ABB RobotStudio station: 1660_smart_tool_trial_final_i_hope - Copy.rsstn

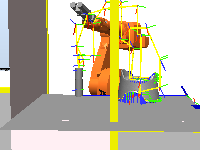
Station 1660_smart_tool_trial_final_i_hope (saved by RobotStudio format 3)
Controller 16-63074
  mechanical unit ROB_1: IRB1600_6_120__02, 6 joints, base frame (0, 0, 0) mm
Layout (positions relative to the parent item):
  - IRB1600_6_120__02 [mechanism, from Robots\IRB1600_6_120__02.rslib] at (0, 0, 0) mm; joint values [-2.0086, -0.3088, 0.1754, -0.2454, -0.2574, 6.5257] (rad or m)
  - Table [part] at (-604.56, -1688.55, 511.81) mm
  - potty-raw7 [part] at (247.23, -520.05, 664.68) mm, rotated rx 89.84 ry 0 rz 0 deg
  - holder [part, from Libraries\holder.rslib] at (-339.39, -762.82, 513.51) mm
  - Dist_to_holder [part] at (-363.16, -741.72, 512.9) mm
  - SmartComponent_1 [smart component] at (-276.35, -599.89, 1043.13) mm, rotated rx -2.86 ry 68.05 rz -114.34 deg
      signals: DI GripperClose, DI GripperOpen
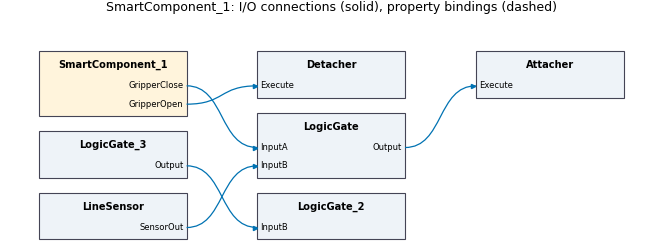
      connections:
        SmartComponent_1.GripperClose -> LogicGate.InputA
        LogicGate.Output -> Attacher.Execute
        LogicGate_3.Output -> LogicGate_2.InputB
        LineSensor.SensorOut -> LogicGate.InputB
        SmartComponent_1.GripperOpen -> Detacher.Execute
    - Kosy_Tool_No_Pen [mechanism] at (0, 0, 0) mm
        TCP Kosy_Tool_No_Pen at (121, 0, 178) mm
        links: tool-m2
    - Attacher [smart component, from Components\Attacher.rslib]
        properties: Parent=Kosy_Tool_No_Pen; Flange=0; Child=tool-m2; Mount=false; Offset=[0 0 0]; Orientation=[0 0 0]
    - Detacher [smart component, from Components\Detacher.rslib]
        properties: Child=tool-m2; KeepPosition=true
    - LogicGate [smart component, from Components\LogicGate.rslib]
        properties: Operator=AND; Delay=0
    - LogicGate_2 [smart component, from Components\LogicGate.rslib]
        properties: Operator=AND; Delay=0
    - LogicGate_3 [smart component, from Components\LogicGate.rslib]
        properties: Operator=NOT; Delay=0
    - LineSensor [smart component, from Components\LineSensor.rslib] at (-8.98, 1.66, 185.12) mm, rotated rx 90 ry 0 rz 90 deg
        properties: Start=[0 0 0]; End=[0 0 0.02]; Radius=0.004; SensedPart=(none); SensedPoint=[0 0 0]
      - _sensorPart_ [part]
  - tool-m2 [part] at (-413.78, -599.19, 679.79) mm, rotated rx -89.18 ry -2.32 rz -154.99 deg
  - Dist_to_backwall [part] at (0, -688.26, 499.44) mm
  - backwall [part] at (-1365.47, 1257.61, -1429.17) mm, rotated rx 90 ry 0 rz 0 deg
  - side wall [part] at (-604.66, -1489.36, -1403.01) mm, rotated rx 90 ry 0 rz 90 deg
  - Dist_to_sidewall2 [part] at (333.28, -1279.39, 533.83) mm
  - sidewall2 [part] at (1386.65, -1478.12, -1427.79) mm, rotated rx 0 ry -90 rz 0 deg
  - Fence_2500 [graphiccomponentgroup, from Equipment\Fence_2500.rslib] at (-617.42, -469.44, -409.13) mm, rotated rx 0 ry 0 rz 90 deg
    - Body 1 [part, from Equipment\Fence_2500.rslib]
    - Body 2 [part, from Equipment\Fence_2500.rslib]
  - bottom [part] at (306.66, -1495.49, -398.13) mm, rotated rx 0 ry -90 rz 90 deg
  - Gate [graphiccomponentgroup, from Equipment\Fence_Gate.rslib] at (-98.47, -1503.2, -434.3) mm, rotated rx 0 ry 0 rz -90 deg
    - Body 1 [part, from Equipment\Fence_Gate.rslib]
    - Body 2 [part, from Equipment\Fence_Gate.rslib]
    - Body 3 [part, from Equipment\Fence_Gate.rslib]
  - ground [part] at (-4365.19, -3484.91, 5.92) mm
Attachment: SmartComponent_1 is attached to IRB1600_6_120__02 / Link6
Collision set CollisionSet_1: SmartComponent_1, tool-m2 against Table, bottom, backwall, Fence_2500, Gate, sidewall2, side wall, near miss 0.005 m
Station logic (signal -> signal, property => property):
  16-63074.OpenGripper -> SmartComponent_1.GripperOpen
  16-63074.CloseGripper -> SmartComponent_1.GripperClose
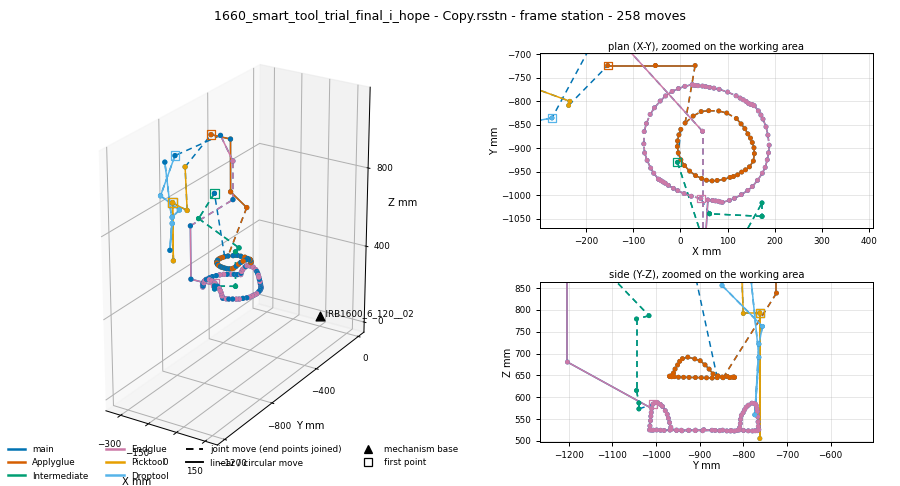
[picture p0: tool path of 1660_smart_tool_trial_final_i_hope - Copy.rsstn in frame station, 258 of 258 moves have a stored position in this frame; points joined in program order, loops and branches not executed]
Targets, tools, work objects and paths stored in the station, written as RAPID:
! task T_ROB1
MODULE MainModule
  TASK PERS tooldata tool1:=[TRUE,[[120.656,0.177793,177.769],[1,0,0,0]],[2,[0,50,88],[1,0,0,0],0,0,0]];
  PROC main()
    MoveJ Target_1290,v600,z100,Kosy_Tool\WObj:=Kosy_wobj;
    MoveJ Target_1210,v600,z100,Kosy_Tool\WObj:=Kosy_wobj;
    WaitTime 1;
    MoveJ Target_1200,v600,z100,Kosy_Tool\WObj:=Kosy_wobj;
    MoveJ Target_1190,v600,z100,Kosy_Tool\WObj:=Kosy_wobj;
    MoveJ Target_1180,v600,z100,Kosy_Tool\WObj:=Kosy_wobj;
    MoveJ Target_360,v600,z100,Kosy_Tool\WObj:=Kosy_wobj;
    MoveL Target_370,v600,z100,Kosy_Tool\WObj:=Kosy_wobj;
    MoveL Target_380,v600,z100,Kosy_Tool\WObj:=Kosy_wobj;
    MoveL Target_390,v600,z100,Kosy_Tool\WObj:=Kosy_wobj;
    MoveJ Target_10,v500,z100,Kosy_Tool\WObj:=Kosy_wobj;
    MoveJ Target_20,v500,z100,Kosy_Tool\WObj:=Kosy_wobj;
    MoveJ Target_30,v500,z100,Kosy_Tool\WObj:=Kosy_wobj;
    MoveJ Target_40,v500,z100,Kosy_Tool\WObj:=Kosy_wobj;
    MoveJ Target_50,v500,z100,Kosy_Tool\WObj:=Kosy_wobj;
    MoveJ Target_60,v500,z100,Kosy_Tool\WObj:=Kosy_wobj;
    MoveJ Target_70,v500,z100,Kosy_Tool\WObj:=Kosy_wobj;
    MoveJ Target_80,v500,z100,Kosy_Tool\WObj:=Kosy_wobj;
    MoveJ Target_90,v500,z100,Kosy_Tool\WObj:=Kosy_wobj;
    MoveJ Target_100,v500,z100,Kosy_Tool\WObj:=Kosy_wobj;
    MoveJ Target_110,v500,z100,Kosy_Tool\WObj:=Kosy_wobj;
    MoveJ Target_120,v500,z100,Kosy_Tool\WObj:=Kosy_wobj;
    MoveJ Target_130,v500,z100,Kosy_Tool\WObj:=Kosy_wobj;
    MoveJ Target_140,v500,z100,Kosy_Tool\WObj:=Kosy_wobj;
    MoveJ Target_150,v500,z100,Kosy_Tool\WObj:=Kosy_wobj;
    MoveJ Target_160,v500,z100,Kosy_Tool\WObj:=Kosy_wobj;
    MoveJ Target_170,v500,z100,Kosy_Tool\WObj:=Kosy_wobj;
    MoveJ Target_180,v500,z100,Kosy_Tool\WObj:=Kosy_wobj;
    MoveJ Target_190,v500,z100,Kosy_Tool\WObj:=Kosy_wobj;
    MoveJ Target_200,v500,z100,Kosy_Tool\WObj:=Kosy_wobj;
    MoveJ Target_210,v500,z100,Kosy_Tool\WObj:=Kosy_wobj;
    MoveJ Target_220,v500,z100,Kosy_Tool\WObj:=Kosy_wobj;
    MoveJ Target_230,v500,z100,Kosy_Tool\WObj:=Kosy_wobj;
    MoveJ Target_240,v500,z100,Kosy_Tool\WObj:=Kosy_wobj;
    MoveJ Target_250,v500,z100,Kosy_Tool\WObj:=Kosy_wobj;
    MoveJ Target_260,v500,z100,Kosy_Tool\WObj:=Kosy_wobj;
    MoveJ Target_270,v500,z100,Kosy_Tool\WObj:=Kosy_wobj;
    MoveJ Target_280,v500,z100,Kosy_Tool\WObj:=Kosy_wobj;
    MoveJ Target_290,v500,z100,Kosy_Tool\WObj:=Kosy_wobj;
    MoveJ Target_300,v500,z100,Kosy_Tool\WObj:=Kosy_wobj;
    MoveJ Target_310,v500,z100,Kosy_Tool\WObj:=Kosy_wobj;
    MoveJ Target_320,v500,z100,Kosy_Tool\WObj:=Kosy_wobj;
    MoveJ Target_330,v500,z100,Kosy_Tool\WObj:=Kosy_wobj;
    MoveJ Target_340,v500,z100,Kosy_Tool\WObj:=Kosy_wobj;
    MoveJ Target_350,v500,z100,Kosy_Tool\WObj:=Kosy_wobj;
    MoveJ Target_400,v600,z100,Kosy_Tool\WObj:=Kosy_wobj;
    MoveJ Target_410,v600,z100,Kosy_Tool\WObj:=Kosy_wobj;
    MoveJ Target_420,v600,z100,Kosy_Tool\WObj:=Kosy_wobj;
    MoveJ Target_430,v600,z100,Kosy_Tool\WObj:=Kosy_wobj;
    MoveJ Target_440,v600,z100,Kosy_Tool\WObj:=Kosy_wobj;
    MoveJ Target_450,v600,z100,Kosy_Tool\WObj:=Kosy_wobj;
    MoveJ Target_460,v600,z100,Kosy_Tool\WObj:=Kosy_wobj;
    MoveJ Target_470,v500,z100,Kosy_Tool\WObj:=Kosy_wobj;
    MoveJ Target_480,v500,z100,Kosy_Tool\WObj:=Kosy_wobj;
    MoveJ Target_490,v500,z100,Kosy_Tool\WObj:=Kosy_wobj;
    MoveJ Target_500,v500,z100,Kosy_Tool\WObj:=Kosy_wobj;
    MoveJ Target_510,v500,z100,Kosy_Tool\WObj:=Kosy_wobj;
    MoveJ Target_520,v500,z100,Kosy_Tool\WObj:=Kosy_wobj;
    MoveJ Target_530,v500,z100,Kosy_Tool\WObj:=Kosy_wobj;
    MoveJ Target_540,v500,z100,Kosy_Tool\WObj:=Kosy_wobj;
    MoveJ Target_550,v500,z100,Kosy_Tool\WObj:=Kosy_wobj;
    MoveJ Target_560,v500,z100,Kosy_Tool\WObj:=Kosy_wobj;
    MoveJ Target_570,v500,z100,Kosy_Tool\WObj:=Kosy_wobj;
    MoveJ Target_580,v500,z100,Kosy_Tool\WObj:=Kosy_wobj;
    MoveJ Target_590,v500,z100,Kosy_Tool\WObj:=Kosy_wobj;
    MoveJ Target_600,v500,z100,Kosy_Tool\WObj:=Kosy_wobj;
    MoveJ Target_610,v500,z100,Kosy_Tool\WObj:=Kosy_wobj;
    MoveJ Target_620,v500,z100,Kosy_Tool\WObj:=Kosy_wobj;
    MoveJ Target_630,v500,z100,Kosy_Tool\WObj:=Kosy_wobj;
    MoveJ Target_640,v500,z100,Kosy_Tool\WObj:=Kosy_wobj;
    MoveJ Target_650,v500,z100,Kosy_Tool\WObj:=Kosy_wobj;
    MoveJ Target_660,v500,z100,Kosy_Tool\WObj:=Kosy_wobj;
    MoveJ Target_670,v500,z100,Kosy_Tool\WObj:=Kosy_wobj;
    MoveJ Target_680,v500,z100,Kosy_Tool\WObj:=Kosy_wobj;
    MoveJ Target_690,v500,z100,Kosy_Tool\WObj:=Kosy_wobj;
    MoveJ Target_700,v500,z100,Kosy_Tool\WObj:=Kosy_wobj;
    MoveJ Target_710,v500,z100,Kosy_Tool\WObj:=Kosy_wobj;
    MoveJ Target_720,v500,z100,Kosy_Tool\WObj:=Kosy_wobj;
    MoveJ Target_730,v500,z100,Kosy_Tool\WObj:=Kosy_wobj;
    MoveJ Target_740,v500,z100,Kosy_Tool\WObj:=Kosy_wobj;
    MoveJ Target_750,v500,z100,Kosy_Tool\WObj:=Kosy_wobj;
    MoveJ Target_760,v500,z100,Kosy_Tool\WObj:=Kosy_wobj;
    MoveJ Target_770,v500,z100,Kosy_Tool\WObj:=Kosy_wobj;
    MoveJ Target_780,v500,z100,Kosy_Tool\WObj:=Kosy_wobj;
    MoveJ Target_790,v500,z100,Kosy_Tool\WObj:=Kosy_wobj;
    MoveJ Target_800,v500,z100,Kosy_Tool\WObj:=Kosy_wobj;
    MoveJ Target_810,v500,z100,Kosy_Tool\WObj:=Kosy_wobj;
    MoveJ Target_820,v500,z100,Kosy_Tool\WObj:=Kosy_wobj;
    MoveJ Target_830,v500,z100,Kosy_Tool\WObj:=Kosy_wobj;
    MoveJ Target_840,v500,z100,Kosy_Tool\WObj:=Kosy_wobj;
    MoveJ Target_850,v500,z100,Kosy_Tool\WObj:=Kosy_wobj;
    MoveJ Target_860,v500,z100,Kosy_Tool\WObj:=Kosy_wobj;
    MoveJ Target_870,v500,z100,Kosy_Tool\WObj:=Kosy_wobj;
    MoveJ Target_880,v500,z100,Kosy_Tool\WObj:=Kosy_wobj;
    MoveJ Target_890,v500,z100,Kosy_Tool\WObj:=Kosy_wobj;
    MoveJ Target_900,v500,z100,Kosy_Tool\WObj:=Kosy_wobj;
    MoveJ Target_910,v500,z100,Kosy_Tool\WObj:=Kosy_wobj;
    MoveJ Target_920,v500,z100,Kosy_Tool\WObj:=Kosy_wobj;
    MoveJ Target_930,v500,z100,Kosy_Tool\WObj:=Kosy_wobj;
    MoveJ Target_940,v500,z100,Kosy_Tool\WObj:=Kosy_wobj;
    MoveJ Target_950,v500,z100,Kosy_Tool\WObj:=Kosy_wobj;
    MoveJ Target_960,v500,z100,Kosy_Tool\WObj:=Kosy_wobj;
    MoveJ Target_970,v500,z100,Kosy_Tool\WObj:=Kosy_wobj;
    MoveJ Target_980,v500,z100,Kosy_Tool\WObj:=Kosy_wobj;
    MoveJ Target_990,v500,z100,Kosy_Tool\WObj:=Kosy_wobj;
    MoveJ Target_1000,v500,z100,Kosy_Tool\WObj:=Kosy_wobj;
    MoveJ Target_1010,v500,z100,Kosy_Tool\WObj:=Kosy_wobj;
    MoveJ Target_1020,v500,z100,Kosy_Tool\WObj:=Kosy_wobj;
    MoveJ Target_1030,v500,z100,Kosy_Tool\WObj:=Kosy_wobj;
    MoveJ Target_1040,v500,z100,Kosy_Tool\WObj:=Kosy_wobj;
    MoveJ Target_1050,v500,z100,Kosy_Tool\WObj:=Kosy_wobj;
    MoveJ Target_1060,v500,z100,Kosy_Tool\WObj:=Kosy_wobj;
    MoveJ Target_1070,v500,z100,Kosy_Tool\WObj:=Kosy_wobj;
    MoveJ Target_1080,v500,z100,Kosy_Tool\WObj:=Kosy_wobj;
    MoveJ Target_1090,v500,z100,Kosy_Tool\WObj:=Kosy_wobj;
    MoveJ Target_1100,v500,z100,Kosy_Tool\WObj:=Kosy_wobj;
    MoveJ Target_1110,v500,z100,Kosy_Tool\WObj:=Kosy_wobj;
    MoveJ Target_1120,v500,z100,Kosy_Tool\WObj:=Kosy_wobj;
    MoveL Target_1130,v600,z100,Kosy_Tool\WObj:=Kosy_wobj;
    MoveL Target_1140,v600,z100,Kosy_Tool\WObj:=Kosy_wobj;
    MoveJ Target_1150,v600,z100,Kosy_Tool\WObj:=Kosy_wobj;
    MoveJ Target_1160,v600,z100,Kosy_Tool\WObj:=Kosy_wobj;
    MoveJ Target_1170,v600,z100,Kosy_Tool\WObj:=Kosy_wobj;
    MoveJ Target_1220,v600,z100,Kosy_Tool\WObj:=Kosy_wobj;
    MoveJ Target_1230,v600,z100,Kosy_Tool\WObj:=Kosy_wobj;
    MoveJ Target_1240,v600,z100,Kosy_Tool\WObj:=Kosy_wobj;
    MoveJ Target_1250,v600,z100,Kosy_Tool\WObj:=Kosy_wobj;
    MoveJ Target_1260,v600,z100,Kosy_Tool\WObj:=Kosy_wobj;
    WaitTime 0.9;
    MoveJ Target_1270,v600,z100,Kosy_Tool\WObj:=Kosy_wobj;
    MoveJ Target_1280,v600,z100,Kosy_Tool\WObj:=Kosy_wobj;
  ENDPROC
ENDMODULE

! task T_ROB1
MODULE Grippers
  PROC CloseGrippers()
    Reset OpenGripper;
    Set CloseGripper;
  ENDPROC
  PROC OpenGrippers()
    Reset CloseGripper;
    Set OpenGripper;
  ENDPROC
ENDMODULE

! task T_ROB1
MODULE CalibData
  PERS tooldata Kosy_Tool:=[TRUE,[[121,0,178],[1,0,0,0]],[2,[10,20,130],[1,0,0,0],0,0,0]];
  TASK PERS wobjdata Kosy_wobj:=[FALSE,TRUE,"",[[0,0,0],[1,0,0,0]],[[401.85011246,-701.374835796,515.862258954],[0.012325857,-0.278428735,-0.003573486,0.960371149]]];
  PERS tooldata Kosy_Tool_No_Pen:=[TRUE,[[121,0,178],[1,0,0,0]],[3,[0,76,77],[1,0,0,0],0,0,0]];
ENDMODULE

! task T_ROB1
MODULE Module1
  CONST robtarget Target_10:=[[258.438803369,151.435734762,318.571021391],[0.699696425,-0.66082153,0.227860096,0.147714575],[-1,-2,1,0],[9E9,9E9,9E9,9E9,9E9,9E9]];
  CONST robtarget Target_20:=[[244.204412094,136.136662782,309.613339311],[0.699696425,-0.66082153,0.227860096,0.147714575],[-1,-2,1,0],[9E9,9E9,9E9,9E9,9E9,9E9]];
  CONST robtarget Target_30:=[[229.298975768,126.244329738,301.863915608],[0.699696425,-0.66082153,0.227860096,0.147714575],[-1,-2,1,0],[9E9,9E9,9E9,9E9,9E9,9E9]];
  CONST robtarget Target_40:=[[216.294982908,124.088037286,292.47562373],[0.699696425,-0.66082153,0.227860096,0.147714575],[-1,-2,1,0],[9E9,9E9,9E9,9E9,9E9,9E9]];
  CONST robtarget Target_50:=[[198.01372253,124.153726611,281.44350419],[0.699696425,-0.66082153,0.227860096,0.147714575],[-1,-2,1,0],[9E9,9E9,9E9,9E9,9E9,9E9]];
  CONST robtarget Target_60:=[[183.663215628,128.206681793,272.238934181],[0.699696425,-0.66082153,0.227860096,0.147714575],[-1,-2,1,0],[9E9,9E9,9E9,9E9,9E9,9E9]];
  CONST robtarget Target_70:=[[165.153419963,139.335396492,262.911181728],[0.699696425,-0.66082153,0.227860096,0.147714575],[-1,-2,1,0],[9E9,9E9,9E9,9E9,9E9,9E9]];
  CONST robtarget Target_80:=[[157.005628518,150.624633227,256.287693133],[0.699696425,-0.66082153,0.227860096,0.147714575],[-1,-2,1,0],[9E9,9E9,9E9,9E9,9E9,9E9]];
  CONST robtarget Target_90:=[[148.581127833,160.466838532,254.286752428],[0.699696425,-0.66082153,0.227860096,0.147714575],[-1,-2,1,0],[9E9,9E9,9E9,9E9,9E9,9E9]];
  CONST robtarget Target_100:=[[140.582494614,171.395954184,254.610852805],[0.699696425,-0.66082153,0.227860096,0.147714575],[-1,-2,1,0],[9E9,9E9,9E9,9E9,9E9,9E9]];
  CONST robtarget Target_110:=[[129.674816508,180.129874926,261.024057423],[0.699696425,-0.66082153,0.227860096,0.147714575],[-1,-2,1,0],[9E9,9E9,9E9,9E9,9E9,9E9]];
  CONST robtarget Target_120:=[[121.014860151,189.288199757,267.147139489],[0.699696425,-0.66082153,0.227860096,0.147714575],[-1,-2,1,0],[9E9,9E9,9E9,9E9,9E9,9E9]];
  CONST robtarget Target_130:=[[112.630891605,200.136293241,273.23351461],[0.699696425,-0.66082153,0.227860096,0.147714575],[-1,-2,0,0],[9E9,9E9,9E9,9E9,9E9,9E9]];
  CONST robtarget Target_140:=[[109.329324411,212.511324177,276.281968307],[0.699696425,-0.66082153,0.227860096,0.147714575],[-1,-2,0,0],[9E9,9E9,9E9,9E9,9E9,9E9]];
  CONST robtarget Target_150:=[[108.645801556,228.355079682,280.874464125],[0.699696425,-0.66082153,0.227860096,0.147714575],[-1,-2,0,0],[9E9,9E9,9E9,9E9,9E9,9E9]];
  CONST robtarget Target_160:=[[117.22096555,240.856009964,282.411868403],[0.699696425,-0.66082153,0.227860096,0.147714575],[-1,-2,0,0],[9E9,9E9,9E9,9E9,9E9,9E9]];
  CONST robtarget Target_170:=[[127.302768884,247.465200223,281.689112647],[0.699696425,-0.66082153,0.227860096,0.147714575],[-1,-2,0,0],[9E9,9E9,9E9,9E9,9E9,9E9]];
  CONST robtarget Target_180:=[[138.537246472,252.55379005,279.00989478],[0.699696425,-0.66082153,0.227860096,0.147714575],[-1,-2,0,0],[9E9,9E9,9E9,9E9,9E9,9E9]];
  CONST robtarget Target_190:=[[150.665726842,258.634767302,275.731771427],[0.699696425,-0.66082153,0.227860096,0.147714575],[-1,-2,1,0],[9E9,9E9,9E9,9E9,9E9,9E9]];
  CONST robtarget Target_200:=[[162.82371969,262.602280432,272.869747889],[0.699696425,-0.66082153,0.227860096,0.147714575],[-1,-2,1,0],[9E9,9E9,9E9,9E9,9E9,9E9]];
  CONST robtarget Target_210:=[[171.55151671,264.707768752,272.940387088],[0.699696425,-0.66082153,0.227860096,0.147714575],[-1,-2,1,0],[9E9,9E9,9E9,9E9,9E9,9E9]];
  CONST robtarget Target_220:=[[183.581930588,269.191831072,277.686906719],[0.699696425,-0.66082153,0.227860096,0.147714575],[-1,-2,1,0],[9E9,9E9,9E9,9E9,9E9,9E9]];
  CONST robtarget Target_230:=[[196.160955655,271.814543333,284.586486039],[0.699696425,-0.66082153,0.227860096,0.147714575],[-1,-2,1,0],[9E9,9E9,9E9,9E9,9E9,9E9]];
  CONST robtarget Target_240:=[[204.934905246,272.97357773,290.966698336],[0.699696425,-0.66082153,0.227860096,0.147714575],[-1,-2,1,0],[9E9,9E9,9E9,9E9,9E9,9E9]];
  CONST robtarget Target_250:=[[215.111177636,271.835081883,297.032635184],[0.699696425,-0.66082153,0.227860096,0.147714575],[-1,-2,1,0],[9E9,9E9,9E9,9E9,9E9,9E9]];
  CONST robtarget Target_260:=[[224.519904076,268.321124256,301.705380789],[0.699696425,-0.66082153,0.227860096,0.147714575],[-1,-2,1,0],[9E9,9E9,9E9,9E9,9E9,9E9]];
  CONST robtarget Target_270:=[[235.384741087,262.576590646,308.694308332],[0.699696425,-0.66082153,0.227860096,0.147714575],[-1,-2,1,0],[9E9,9E9,9E9,9E9,9E9,9E9]];
  CONST robtarget Target_280:=[[246.907584253,253.329236086,314.436979725],[0.699696425,-0.66082153,0.227860096,0.147714575],[-1,-2,1,0],[9E9,9E9,9E9,9E9,9E9,9E9]];
  CONST robtarget Target_290:=[[256.605146154,241.898819064,320.136202767],[0.699696425,-0.66082153,0.227860096,0.147714575],[-1,-2,1,0],[9E9,9E9,9E9,9E9,9E9,9E9]];
  CONST robtarget Target_300:=[[263.670421532,229.596602909,324.070288514],[0.699696425,-0.66082153,0.227860096,0.147714575],[-1,-2,1,0],[9E9,9E9,9E9,9E9,9E9,9E9]];
  CONST robtarget Target_310:=[[268.773730103,215.083881477,326.794181912],[0.699696425,-0.66082153,0.227860096,0.147714575],[-1,-2,1,0],[9E9,9E9,9E9,9E9,9E9,9E9]];
  CONST robtarget Target_320:=[[271.002990828,201.612792794,327.531776458],[0.699696425,-0.66082153,0.227860096,0.147714575],[-1,-2,1,0],[9E9,9E9,9E9,9E9,9E9,9E9]];
  CONST robtarget Target_330:=[[271.094895998,189.658760325,327.02572338],[0.699696425,-0.66082153,0.227860096,0.147714575],[-1,-2,1,0],[9E9,9E9,9E9,9E9,9E9,9E9]];
  CONST robtarget Target_340:=[[269.248568204,176.721249058,325.065236991],[0.699696425,-0.66082153,0.227860096,0.147714575],[-1,-2,1,0],[9E9,9E9,9E9,9E9,9E9,9E9]];
  CONST robtarget Target_350:=[[265.702454413,165.05754945,323.555757097],[0.699696425,-0.66082153,0.227860096,0.147714575],[-1,-2,1,0],[9E9,9E9,9E9,9E9,9E9,9E9]];
  CONST robtarget Target_360:=[[132.420110035,25.905846589,830.128212546],[0.875109539,-0.297215415,0.097995159,0.36911142],[-2,-2,1,0],[9E9,9E9,9E9,9E9,9E9,9E9]];
  CONST robtarget Target_370:=[[46.786821326,23.707351638,775.900690346],[0.875109552,-0.297215434,0.097995104,0.369111388],[-1,-2,1,0],[9E9,9E9,9E9,9E9,9E9,9E9]];
  CONST robtarget Target_380:=[[180.832304643,27.148762522,564.083557965],[0.875109514,-0.297215484,0.097995119,0.369111436],[-1,-2,1,0],[9E9,9E9,9E9,9E9,9E9,9E9]];
  CONST robtarget Target_390:=[[139.897197574,26.097877718,470.955764332],[0.87510953,-0.297215516,0.097995198,0.369111349],[-1,-2,1,0],[9E9,9E9,9E9,9E9,9E9,9E9]];
  CONST robtarget Target_400:=[[95.744268647,230.654466585,602.666874086],[0.780533546,-0.55853965,0.126987162,0.250349961],[-1,-2,1,0],[9E9,9E9,9E9,9E9,9E9,9E9]];
  CONST robtarget Target_410:=[[20.982247532,485.602413443,552.300858265],[0.640673815,-0.476988614,0.317134258,0.51131672],[-1,-2,1,0],[9E9,9E9,9E9,9E9,9E9,9E9]];
  CONST robtarget Target_420:=[[40.057840571,315.485164605,351.175017316],[0.240330351,-0.75280002,0.602336649,0.11280077],[-1,-2,1,0],[9E9,9E9,9E9,9E9,9E9,9E9]];
  CONST robtarget Target_430:=[[43.325363118,344.238603306,344.849218674],[0.240330216,-0.752800029,0.60233668,0.112800831],[-1,0,0,0],[9E9,9E9,9E9,9E9,9E9,9E9]];
  CONST robtarget Target_440:=[[130.902145722,346.486980546,206.461369243],[0.240330202,-0.752799969,0.602336751,0.112800882],[-1,0,0,0],[9E9,9E9,9E9,9E9,9E9,9E9]];
  CONST robtarget Target_450:=[[240.371318881,343.833384772,242.072398526],[0.349848139,-0.771235082,0.529354347,-0.050859638],[-1,0,-1,0],[9E9,9E9,9E9,9E9,9E9,9E9]];
  CONST robtarget Target_460:=[[247.719237938,344.02203137,230.461334982],[0.349848132,-0.771235147,0.529354256,-0.050859653],[-1,-1,-1,0],[9E9,9E9,9E9,9E9,9E9,9E9]];
  CONST robtarget Target_470:=[[258.409448537,311.900373735,249.670518456],[0.324640606,-0.795683306,0.494988307,-0.128386639],[-1,-1,-1,0],[9E9,9E9,9E9,9E9,9E9,9E9]];
  CONST robtarget Target_480:=[[273.456551263,307.386812239,263.76798686],[0.324640606,-0.795683306,0.494988307,-0.128386639],[-1,-1,-1,0],[9E9,9E9,9E9,9E9,9E9,9E9]];
  CONST robtarget Target_490:=[[286.976995459,302.126853412,271.343159171],[0.324640606,-0.795683306,0.494988307,-0.128386639],[-1,-1,-1,0],[9E9,9E9,9E9,9E9,9E9,9E9]];
  CONST robtarget Target_500:=[[300.6702416,296.165654178,275.45847733],[0.324640606,-0.795683306,0.494988307,-0.128386639],[-1,-1,-1,0],[9E9,9E9,9E9,9E9,9E9,9E9]];
  CONST robtarget Target_510:=[[311.008540577,291.585114548,276.393513506],[0.334594883,-0.749514417,0.562453097,-0.099603796],[-1,-1,-1,0],[9E9,9E9,9E9,9E9,9E9,9E9]];
  CONST robtarget Target_520:=[[325.355626927,285.595642682,273.963195097],[0.342002692,-0.697641271,0.625637279,-0.070062908],[-1,-1,-1,0],[9E9,9E9,9E9,9E9,9E9,9E9]];
  CONST robtarget Target_530:=[[335.497747996,281.316441875,270.385596862],[0.342002692,-0.697641271,0.625637279,-0.070062908],[-2,-1,0,0],[9E9,9E9,9E9,9E9,9E9,9E9]];
  CONST robtarget Target_540:=[[344.250400056,278.950575237,265.097340819],[0.342002692,-0.697641271,0.625637279,-0.070062908],[-2,-1,0,0],[9E9,9E9,9E9,9E9,9E9,9E9]];
  CONST robtarget Target_550:=[[353.307020648,276.450436828,259.127292761],[0.405107701,-0.641506769,0.65123065,0.01598302],[-2,-1,0,0],[9E9,9E9,9E9,9E9,9E9,9E9]];
  CONST robtarget Target_560:=[[362.727197307,273.903094879,252.525484203],[0.40925638,-0.527537431,0.733405691,0.127787191],[-2,-1,0,0],[9E9,9E9,9E9,9E9,9E9,9E9]];
  CONST robtarget Target_570:=[[366.594480317,273.370153015,249.121220136],[0.408894597,-0.609853011,0.678288905,0.028437203],[-2,-1,0,0],[9E9,9E9,9E9,9E9,9E9,9E9]];
  CONST robtarget Target_580:=[[376.050602806,261.07345192,252.980640611],[0.450267636,-0.431135604,0.7743672,0.108335526],[-2,-1,0,0],[9E9,9E9,9E9,9E9,9E9,9E9]];
  CONST robtarget Target_590:=[[382.015093252,250.299701272,256.1607371],[0.466856546,-0.373006487,0.797430741,0.083757621],[-2,-1,0,0],[9E9,9E9,9E9,9E9,9E9,9E9]];
  CONST robtarget Target_600:=[[388.783208198,234.076946083,260.157953423],[0.466856546,-0.373006487,0.797430741,0.083757621],[-2,-1,0,0],[9E9,9E9,9E9,9E9,9E9,9E9]];
  CONST robtarget Target_610:=[[394.194307242,218.416777781,262.285988503],[0.466856546,-0.373006487,0.797430741,0.083757621],[-2,-1,0,0],[9E9,9E9,9E9,9E9,9E9,9E9]];
  CONST robtarget Target_620:=[[394.986127271,199.225516918,264.98681791],[0.466856546,-0.373006487,0.797430741,0.083757621],[-2,-1,0,0],[9E9,9E9,9E9,9E9,9E9,9E9]];
  CONST robtarget Target_630:=[[395.808228308,173.082792274,263.21414143],[0.502132199,-0.111207526,0.856866655,0.035716606],[-2,-1,0,0],[9E9,9E9,9E9,9E9,9E9,9E9]];
  CONST robtarget Target_640:=[[392.096007692,155.915946572,261.177916089],[0.484626403,0.085654893,0.861207372,0.126973819],[-2,-1,0,0],[9E9,9E9,9E9,9E9,9E9,9E9]];
  CONST robtarget Target_650:=[[386.23356341,136.300470266,256.168930799],[0.478322069,0.124838154,0.857148411,0.1446376],[-2,-1,1,0],[9E9,9E9,9E9,9E9,9E9,9E9]];
  CONST robtarget Target_660:=[[378.688426604,122.054465472,251.624453686],[0.515255101,0.131028339,0.83546848,0.139054573],[-2,-1,1,0],[9E9,9E9,9E9,9E9,9E9,9E9]];
  CONST robtarget Target_670:=[[368.90918858,107.461824351,244.869240948],[0.501155051,0.186058759,0.837247454,0.115075861],[-2,-1,1,0],[9E9,9E9,9E9,9E9,9E9,9E9]];
  CONST robtarget Target_680:=[[359.87814797,96.376601372,238.096653854],[0.516556654,0.250217693,0.814623329,0.083361628],[-2,-1,1,0],[9E9,9E9,9E9,9E9,9E9,9E9]];
  CONST robtarget Target_690:=[[348.496527259,86.495669296,230.343772866],[0.446373625,0.5584739,0.696370195,0.062658138],[-1,-1,1,0],[9E9,9E9,9E9,9E9,9E9,9E9]];
  CONST robtarget Target_700:=[[337.162767535,80.121148867,223.573598178],[0.448722769,0.670696452,0.588031474,0.055073873],[-1,-1,1,0],[9E9,9E9,9E9,9E9,9E9,9E9]];
  CONST robtarget Target_710:=[[325.683925345,75.07970879,216.390359497],[0.448722769,0.670696452,0.588031474,0.055073873],[-1,-1,2,0],[9E9,9E9,9E9,9E9,9E9,9E9]];
  CONST robtarget Target_720:=[[311.152675753,71.01170282,210.209203801],[0.448722769,0.670696452,0.588031474,0.055073873],[-1,-1,2,0],[9E9,9E9,9E9,9E9,9E9,9E9]];
  CONST robtarget Target_730:=[[305.690093339,72.022841225,215.697132848],[0.387401332,0.699269705,0.596859221,0.068564992],[-1,-1,2,0],[9E9,9E9,9E9,9E9,9E9,9E9]];
  CONST robtarget Target_740:=[[296.55914547,72.334438069,222.002911323],[0.387401332,0.699269705,0.596859221,0.068564992],[-1,-1,2,0],[9E9,9E9,9E9,9E9,9E9,9E9]];
  CONST robtarget Target_750:=[[285.03551515,72.732238797,228.484093174],[0.387401332,0.699269705,0.596859221,0.068564992],[-1,-1,2,0],[9E9,9E9,9E9,9E9,9E9,9E9]];
  CONST robtarget Target_760:=[[270.716548642,73.111392456,233.394273074],[0.387401332,0.699269705,0.596859221,0.068564992],[-1,-1,2,0],[9E9,9E9,9E9,9E9,9E9,9E9]];
  CONST robtarget Target_770:=[[261.257990589,74.11390554,235.540526075],[0.387401332,0.699269705,0.596859221,0.068564992],[-1,-1,2,0],[9E9,9E9,9E9,9E9,9E9,9E9]];
  CONST robtarget Target_780:=[[250.354210611,75.422079463,237.166947393],[0.387401332,0.699269705,0.596859221,0.068564992],[-1,-1,2,0],[9E9,9E9,9E9,9E9,9E9,9E9]];
  CONST robtarget Target_790:=[[240.888321632,76.770404541,234.883956846],[0.387401332,0.699269705,0.596859221,0.068564992],[-1,-1,2,0],[9E9,9E9,9E9,9E9,9E9,9E9]];
  CONST robtarget Target_800:=[[230.571222825,78.965448595,230.224829128],[0.387401332,0.699269705,0.596859221,0.068564992],[-1,-1,2,0],[9E9,9E9,9E9,9E9,9E9,9E9]];
  CONST robtarget Target_810:=[[214.903451101,84.385437473,221.04109893],[0.387401332,0.699269705,0.596859221,0.068564992],[-1,-1,2,0],[9E9,9E9,9E9,9E9,9E9,9E9]];
  CONST robtarget Target_820:=[[201.988283762,91.996421769,207.572856595],[0.387401332,0.699269705,0.596859221,0.068564992],[-1,-1,2,0],[9E9,9E9,9E9,9E9,9E9,9E9]];
  CONST robtarget Target_830:=[[196.892410546,96.767477733,199.306011126],[0.387401332,0.699269705,0.596859221,0.068564992],[-1,-1,2,0],[9E9,9E9,9E9,9E9,9E9,9E9]];
  CONST robtarget Target_840:=[[194.316463311,100.329187929,190.746530058],[0.387401332,0.699269705,0.596859221,0.068564992],[-1,0,2,0],[9E9,9E9,9E9,9E9,9E9,9E9]];
  CONST robtarget Target_850:=[[192.775639617,103.840299173,181.479695304],[0.36960965,0.792289743,0.466364678,0.134794871],[-1,0,2,0],[9E9,9E9,9E9,9E9,9E9,9E9]];
  CONST robtarget Target_860:=[[191.850239876,107.963048659,173.569689381],[0.375137533,0.771193117,0.500479995,0.11854443],[-1,0,2,0],[9E9,9E9,9E9,9E9,9E9,9E9]];
  CONST robtarget Target_870:=[[193.299045608,109.853271468,163.782694284],[0.375137533,0.771193117,0.500479995,0.11854443],[-1,0,2,0],[9E9,9E9,9E9,9E9,9E9,9E9]];
  CONST robtarget Target_880:=[[195.510685576,110.371812275,154.144459973],[0.318618532,0.828336835,0.456811969,0.060523909],[-1,0,2,0],[9E9,9E9,9E9,9E9,9E9,9E9]];
  CONST robtarget Target_890:=[[197.804086033,111.862864553,144.843138708],[0.318618532,0.828336835,0.456811969,0.060523909],[-1,0,2,0],[9E9,9E9,9E9,9E9,9E9,9E9]];
  CONST robtarget Target_900:=[[199.19793959,113.006863358,138.921816404],[0.204531401,0.919028423,0.336422513,0.019327606],[-1,0,2,0],[9E9,9E9,9E9,9E9,9E9,9E9]];
  CONST robtarget Target_910:=[[192.895853489,123.902605126,132.209324541],[0.157383635,0.953791608,0.253268199,0.036975378],[-1,0,2,0],[9E9,9E9,9E9,9E9,9E9,9E9]];
  CONST robtarget Target_920:=[[187.9708826,132.586074252,129.452005105],[0.125396201,-0.991266326,-0.039779352,0.009190602],[-1,0,2,0],[9E9,9E9,9E9,9E9,9E9,9E9]];
  CONST robtarget Target_930:=[[183.909913207,141.095432354,127.220352246],[0.132897256,-0.988676587,-0.069687184,0.000788619],[-1,0,2,0],[9E9,9E9,9E9,9E9,9E9,9E9]];
  CONST robtarget Target_940:=[[177.824514971,157.308484399,124.134535201],[0.250167727,-0.967041618,0.034649248,-0.032342651],[-1,0,2,0],[9E9,9E9,9E9,9E9,9E9,9E9]];
  CONST robtarget Target_950:=[[173.394741319,174.789237632,122.913032769],[0.251840312,-0.946030749,0.200406693,-0.03793992],[-1,0,3,0],[9E9,9E9,9E9,9E9,9E9,9E9]];
  CONST robtarget Target_960:=[[171.180085409,196.127367201,120.498624847],[0.213782262,-0.96447622,0.154571079,-0.013803875],[-1,0,3,0],[9E9,9E9,9E9,9E9,9E9,9E9]];
  CONST robtarget Target_970:=[[171.225439064,212.447444508,122.386819819],[0.398152545,-0.909634863,0.118246125,-0.00753791],[-1,0,3,0],[9E9,9E9,9E9,9E9,9E9,9E9]];
  CONST robtarget Target_980:=[[173.306878849,227.367534017,123.387176518],[0.383105424,-0.908447481,0.155845573,-0.060543917],[-1,0,3,0],[9E9,9E9,9E9,9E9,9E9,9E9]];
  CONST robtarget Target_990:=[[177.176148055,243.621727869,124.889466949],[0.363446291,-0.89736073,0.238943407,-0.07454235],[-1,-1,3,0],[9E9,9E9,9E9,9E9,9E9,9E9]];
  CONST robtarget Target_1000:=[[181.623159332,256.114241681,128.79871545],[0.352569269,-0.889248994,0.279849428,-0.081335323],[-1,-1,3,0],[9E9,9E9,9E9,9E9,9E9,9E9]];
  CONST robtarget Target_1010:=[[189.320003001,271.333271532,134.951107186],[0.347631525,-0.88769406,0.285959987,-0.09684247],[-1,-1,3,0],[9E9,9E9,9E9,9E9,9E9,9E9]];
  CONST robtarget Target_1020:=[[198.779444868,285.01695411,140.10381253],[0.335380516,-0.87777523,0.326125606,-0.103308494],[-1,-1,3,0],[9E9,9E9,9E9,9E9,9E9,9E9]];
  CONST robtarget Target_1030:=[[206.561512747,293.298263909,145.776423498],[0.350101384,-0.801312087,0.477319566,-0.086567843],[-1,-1,3,0],[9E9,9E9,9E9,9E9,9E9,9E9]];
  CONST robtarget Target_1040:=[[217.428774095,302.557025511,153.57553574],[0.350101384,-0.801312087,0.477319566,-0.086567843],[-1,-1,3,0],[9E9,9E9,9E9,9E9,9E9,9E9]];
  CONST robtarget Target_1050:=[[229.963623987,310.920424163,161.086033851],[0.350101384,-0.801312087,0.477319566,-0.086567843],[-1,-1,3,0],[9E9,9E9,9E9,9E9,9E9,9E9]];
  CONST robtarget Target_1060:=[[238.770788693,315.270204795,166.800265656],[0.362476182,-0.80330358,0.467991415,-0.065562273],[-1,-1,3,0],[9E9,9E9,9E9,9E9,9E9,9E9]];
  CONST robtarget Target_1070:=[[251.089382176,319.789995238,175.404432124],[0.364068191,-0.790777721,0.488859082,-0.056051286],[-1,-1,3,0],[9E9,9E9,9E9,9E9,9E9,9E9]];
  CONST robtarget Target_1080:=[[250.070385456,318.848615897,185.722424785],[0.364068191,-0.790777721,0.488859082,-0.056051286],[-1,-1,3,0],[9E9,9E9,9E9,9E9,9E9,9E9]];
  CONST robtarget Target_1090:=[[247.223293569,317.411913667,197.781435257],[0.364068191,-0.790777721,0.488859082,-0.056051286],[-1,-1,3,0],[9E9,9E9,9E9,9E9,9E9,9E9]];
  CONST robtarget Target_1100:=[[246.793575015,316.610093603,209.491636447],[0.364068191,-0.790777721,0.488859082,-0.056051286],[-1,-1,3,0],[9E9,9E9,9E9,9E9,9E9,9E9]];
  CONST robtarget Target_1110:=[[247.393446991,315.711313699,220.283270251],[0.365410686,-0.777709902,0.50939171,-0.046501885],[-1,-1,3,0],[9E9,9E9,9E9,9E9,9E9,9E9]];
  CONST robtarget Target_1120:=[[250.961262817,314.648416801,233.354047647],[0.366502746,-0.76410908,0.529575226,-0.036920613],[-1,-1,3,0],[9E9,9E9,9E9,9E9,9E9,9E9]];
  CONST robtarget Target_1130:=[[198.735913663,506.382233448,329.120791713],[0.614984275,-0.678796732,0.334169216,0.22217172],[-1,-1,4,0],[9E9,9E9,9E9,9E9,9E9,9E9]];
  CONST robtarget Target_1140:=[[65.537479642,502.962797939,539.599274694],[0.614984197,-0.678796732,0.334169309,0.222171796],[-1,-1,3,0],[9E9,9E9,9E9,9E9,9E9,9E9]];
  CONST robtarget Target_1150:=[[74.234698422,164.194273086,539.599263219],[0.614984131,-0.678796816,0.334169273,0.222171776],[-1,-1,3,0],[9E9,9E9,9E9,9E9,9E9,9E9]];
  CONST robtarget Target_1160:=[[-22.605648694,161.708068633,692.625267245],[0.614984163,-0.678796806,0.334169252,0.222171749],[-1,-1,4,0],[9E9,9E9,9E9,9E9,9E9,9E9]];
  CONST robtarget Target_1170:=[[161.190855274,-64.987192787,805.255214948],[0.614984123,-0.678796828,0.334169258,0.222171783],[-2,0,3,0],[9E9,9E9,9E9,9E9,9E9,9E9]];
  CONST robtarget Target_1180:=[[276.182354787,114.471258764,754.716801553],[0.735359782,-0.488406919,0.300048701,0.361490594],[-2,-2,1,0],[9E9,9E9,9E9,9E9,9E9,9E9]];
  CONST robtarget Target_1190:=[[387.744774333,108.48003588,573.904245654],[0.693177998,-0.528527986,0.38979131,0.297027213],[-2,-2,1,0],[9E9,9E9,9E9,9E9,9E9,9E9]];
  CONST robtarget Target_1200:=[[475.906525543,72.848154714,629.117273062],[0.726504015,-0.480945745,0.408546632,0.271979329],[-2,-2,1,0],[9E9,9E9,9E9,9E9,9E9,9E9]];
  CONST robtarget Target_1210:=[[629.010784483,76.778825732,387.183728782],[0.726503998,-0.48094574,0.408546657,0.271979345],[-2,-2,2,0],[9E9,9E9,9E9,9E9,9E9,9E9]];
  CONST robtarget Target_1220:=[[275.931265647,141.060107315,820.144257615],[0.718245148,-0.523288771,0.361402039,0.282278825],[-2,-1,3,0],[9E9,9E9,9E9,9E9,9E9,9E9]];
  CONST robtarget Target_1230:=[[444.606550427,158.67603468,686.660199071],[0.728174977,-0.506340379,0.380953951,0.261256023],[-2,-1,3,0],[9E9,9E9,9E9,9E9,9E9,9E9]];
  CONST robtarget Target_1240:=[[464.56080754,66.530963056,586.899667272],[0.736558505,-0.500901623,0.362113056,0.274687583],[-2,-1,3,1],[9E9,9E9,9E9,9E9,9E9,9E9]];
  CONST robtarget Target_1250:=[[515.159875493,75.954926124,571.115734521],[0.72539825,-0.49351912,0.383574371,0.288282777],[-2,-1,4,1],[9E9,9E9,9E9,9E9,9E9,9E9]];
  CONST robtarget Target_1260:=[[608.496672526,87.854326358,438.664859678],[0.720516306,-0.494692804,0.391893041,0.287324079],[-2,-1,4,1],[9E9,9E9,9E9,9E9,9E9,9E9]];
  CONST robtarget Target_1270:=[[531.419901202,76.372365213,545.421913323],[0.72539833,-0.493519128,0.383574254,0.288282717],[-2,-1,4,1],[9E9,9E9,9E9,9E9,9E9,9E9]];
  CONST robtarget Target_1280:=[[379.301456663,103.387507022,811.593803105],[0.784581809,-0.439434545,0.243282767,0.363513634],[-2,-1,4,1],[9E9,9E9,9E9,9E9,9E9,9E9]];
  CONST robtarget Target_1290:=[[475.049509691,72.826158816,630.471496488],[0.726504,-0.480945723,0.408546658,0.271979371],[-2,-2,1,0],[9E9,9E9,9E9,9E9,9E9,9E9]];
  PROC Applyglue()
    MoveJ Target_360,v600,z100,Kosy_Tool\WObj:=Kosy_wobj;
    MoveL Target_370,v600,z100,Kosy_Tool\WObj:=Kosy_wobj;
    MoveL Target_380,v600,z100,Kosy_Tool\WObj:=Kosy_wobj;
    MoveL Target_390,v600,z100,Kosy_Tool\WObj:=Kosy_wobj;
    MoveJ Target_10,v500,z100,Kosy_Tool\WObj:=Kosy_wobj;
    MoveJ Target_20,v500,z100,Kosy_Tool\WObj:=Kosy_wobj;
    MoveJ Target_30,v500,z100,Kosy_Tool\WObj:=Kosy_wobj;
    MoveJ Target_40,v500,z100,Kosy_Tool\WObj:=Kosy_wobj;
    MoveJ Target_50,v500,z100,Kosy_Tool\WObj:=Kosy_wobj;
    MoveJ Target_60,v500,z100,Kosy_Tool\WObj:=Kosy_wobj;
    MoveJ Target_70,v500,z100,Kosy_Tool\WObj:=Kosy_wobj;
    MoveJ Target_80,v500,z100,Kosy_Tool\WObj:=Kosy_wobj;
    MoveJ Target_90,v500,z100,Kosy_Tool\WObj:=Kosy_wobj;
    MoveJ Target_100,v500,z100,Kosy_Tool\WObj:=Kosy_wobj;
    MoveJ Target_110,v500,z100,Kosy_Tool\WObj:=Kosy_wobj;
    MoveJ Target_120,v500,z100,Kosy_Tool\WObj:=Kosy_wobj;
    MoveJ Target_130,v500,z100,Kosy_Tool\WObj:=Kosy_wobj;
    MoveJ Target_140,v500,z100,Kosy_Tool\WObj:=Kosy_wobj;
    MoveJ Target_150,v500,z100,Kosy_Tool\WObj:=Kosy_wobj;
    MoveJ Target_160,v500,z100,Kosy_Tool\WObj:=Kosy_wobj;
    MoveJ Target_170,v500,z100,Kosy_Tool\WObj:=Kosy_wobj;
    MoveJ Target_180,v500,z100,Kosy_Tool\WObj:=Kosy_wobj;
    MoveJ Target_190,v500,z100,Kosy_Tool\WObj:=Kosy_wobj;
    MoveJ Target_200,v500,z100,Kosy_Tool\WObj:=Kosy_wobj;
    MoveJ Target_210,v500,z100,Kosy_Tool\WObj:=Kosy_wobj;
    MoveJ Target_220,v500,z100,Kosy_Tool\WObj:=Kosy_wobj;
    MoveJ Target_230,v500,z100,Kosy_Tool\WObj:=Kosy_wobj;
    MoveJ Target_240,v500,z100,Kosy_Tool\WObj:=Kosy_wobj;
    MoveJ Target_250,v500,z100,Kosy_Tool\WObj:=Kosy_wobj;
    MoveJ Target_260,v500,z100,Kosy_Tool\WObj:=Kosy_wobj;
    MoveJ Target_270,v500,z100,Kosy_Tool\WObj:=Kosy_wobj;
    MoveJ Target_280,v500,z100,Kosy_Tool\WObj:=Kosy_wobj;
    MoveJ Target_290,v500,z100,Kosy_Tool\WObj:=Kosy_wobj;
    MoveJ Target_300,v500,z100,Kosy_Tool\WObj:=Kosy_wobj;
    MoveJ Target_310,v500,z100,Kosy_Tool\WObj:=Kosy_wobj;
    MoveJ Target_320,v500,z100,Kosy_Tool\WObj:=Kosy_wobj;
    MoveJ Target_330,v500,z100,Kosy_Tool\WObj:=Kosy_wobj;
    MoveJ Target_340,v500,z100,Kosy_Tool\WObj:=Kosy_wobj;
    MoveJ Target_350,v500,z100,Kosy_Tool\WObj:=Kosy_wobj;
  ENDPROC
  PROC Intermediate()
    MoveJ Target_400,v600,z100,Kosy_Tool\WObj:=Kosy_wobj;
    MoveJ Target_410,v600,z100,Kosy_Tool\WObj:=Kosy_wobj;
    MoveJ Target_420,v600,z100,Kosy_Tool\WObj:=Kosy_wobj;
    MoveJ Target_430,v600,z100,Kosy_Tool\WObj:=Kosy_wobj;
    MoveJ Target_440,v600,z100,Kosy_Tool\WObj:=Kosy_wobj;
    MoveJ Target_450,v600,z100,Kosy_Tool\WObj:=Kosy_wobj;
    MoveJ Target_460,v600,z100,Kosy_Tool\WObj:=Kosy_wobj;
  ENDPROC
  PROC Endglue()
    MoveJ Target_470,v500,z100,Kosy_Tool\WObj:=Kosy_wobj;
    MoveJ Target_480,v500,z100,Kosy_Tool\WObj:=Kosy_wobj;
    MoveJ Target_490,v500,z100,Kosy_Tool\WObj:=Kosy_wobj;
    MoveJ Target_500,v500,z100,Kosy_Tool\WObj:=Kosy_wobj;
    MoveJ Target_510,v500,z100,Kosy_Tool\WObj:=Kosy_wobj;
    MoveJ Target_520,v500,z100,Kosy_Tool\WObj:=Kosy_wobj;
    MoveJ Target_530,v500,z100,Kosy_Tool\WObj:=Kosy_wobj;
    MoveJ Target_540,v500,z100,Kosy_Tool\WObj:=Kosy_wobj;
    MoveJ Target_550,v500,z100,Kosy_Tool\WObj:=Kosy_wobj;
    MoveJ Target_560,v500,z100,Kosy_Tool\WObj:=Kosy_wobj;
    MoveJ Target_570,v500,z100,Kosy_Tool\WObj:=Kosy_wobj;
    MoveJ Target_580,v500,z100,Kosy_Tool\WObj:=Kosy_wobj;
    MoveJ Target_590,v500,z100,Kosy_Tool\WObj:=Kosy_wobj;
    MoveJ Target_600,v500,z100,Kosy_Tool\WObj:=Kosy_wobj;
    MoveJ Target_610,v500,z100,Kosy_Tool\WObj:=Kosy_wobj;
    MoveJ Target_620,v500,z100,Kosy_Tool\WObj:=Kosy_wobj;
    MoveJ Target_630,v500,z100,Kosy_Tool\WObj:=Kosy_wobj;
    MoveJ Target_640,v500,z100,Kosy_Tool\WObj:=Kosy_wobj;
    MoveJ Target_650,v500,z100,Kosy_Tool\WObj:=Kosy_wobj;
    MoveJ Target_660,v500,z100,Kosy_Tool\WObj:=Kosy_wobj;
    MoveJ Target_670,v500,z100,Kosy_Tool\WObj:=Kosy_wobj;
    MoveJ Target_680,v500,z100,Kosy_Tool\WObj:=Kosy_wobj;
    MoveJ Target_690,v500,z100,Kosy_Tool\WObj:=Kosy_wobj;
    MoveJ Target_700,v500,z100,Kosy_Tool\WObj:=Kosy_wobj;
    MoveJ Target_710,v500,z100,Kosy_Tool\WObj:=Kosy_wobj;
    MoveJ Target_720,v500,z100,Kosy_Tool\WObj:=Kosy_wobj;
    MoveJ Target_730,v500,z100,Kosy_Tool\WObj:=Kosy_wobj;
    MoveJ Target_740,v500,z100,Kosy_Tool\WObj:=Kosy_wobj;
    MoveJ Target_750,v500,z100,Kosy_Tool\WObj:=Kosy_wobj;
    MoveJ Target_760,v500,z100,Kosy_Tool\WObj:=Kosy_wobj;
    MoveJ Target_770,v500,z100,Kosy_Tool\WObj:=Kosy_wobj;
    MoveJ Target_780,v500,z100,Kosy_Tool\WObj:=Kosy_wobj;
    MoveJ Target_790,v500,z100,Kosy_Tool\WObj:=Kosy_wobj;
    MoveJ Target_800,v500,z100,Kosy_Tool\WObj:=Kosy_wobj;
    MoveJ Target_810,v500,z100,Kosy_Tool\WObj:=Kosy_wobj;
    MoveJ Target_820,v500,z100,Kosy_Tool\WObj:=Kosy_wobj;
    MoveJ Target_830,v500,z100,Kosy_Tool\WObj:=Kosy_wobj;
    MoveJ Target_840,v500,z100,Kosy_Tool\WObj:=Kosy_wobj;
    MoveJ Target_850,v500,z100,Kosy_Tool\WObj:=Kosy_wobj;
    MoveJ Target_860,v500,z100,Kosy_Tool\WObj:=Kosy_wobj;
    MoveJ Target_870,v500,z100,Kosy_Tool\WObj:=Kosy_wobj;
    MoveJ Target_880,v500,z100,Kosy_Tool\WObj:=Kosy_wobj;
    MoveJ Target_890,v500,z100,Kosy_Tool\WObj:=Kosy_wobj;
    MoveJ Target_900,v500,z100,Kosy_Tool\WObj:=Kosy_wobj;
    MoveJ Target_910,v500,z100,Kosy_Tool\WObj:=Kosy_wobj;
    MoveJ Target_920,v500,z100,Kosy_Tool\WObj:=Kosy_wobj;
    MoveJ Target_930,v500,z100,Kosy_Tool\WObj:=Kosy_wobj;
    MoveJ Target_940,v500,z100,Kosy_Tool\WObj:=Kosy_wobj;
    MoveJ Target_950,v500,z100,Kosy_Tool\WObj:=Kosy_wobj;
    MoveJ Target_960,v500,z100,Kosy_Tool\WObj:=Kosy_wobj;
    MoveJ Target_970,v500,z100,Kosy_Tool\WObj:=Kosy_wobj;
    MoveJ Target_980,v500,z100,Kosy_Tool\WObj:=Kosy_wobj;
    MoveJ Target_990,v500,z100,Kosy_Tool\WObj:=Kosy_wobj;
    MoveJ Target_1000,v500,z100,Kosy_Tool\WObj:=Kosy_wobj;
    MoveJ Target_1010,v500,z100,Kosy_Tool\WObj:=Kosy_wobj;
    MoveJ Target_1020,v500,z100,Kosy_Tool\WObj:=Kosy_wobj;
    MoveJ Target_1030,v500,z100,Kosy_Tool\WObj:=Kosy_wobj;
    MoveJ Target_1040,v500,z100,Kosy_Tool\WObj:=Kosy_wobj;
    MoveJ Target_1050,v500,z100,Kosy_Tool\WObj:=Kosy_wobj;
    MoveJ Target_1060,v500,z100,Kosy_Tool\WObj:=Kosy_wobj;
    MoveJ Target_1070,v500,z100,Kosy_Tool\WObj:=Kosy_wobj;
    MoveJ Target_1080,v500,z100,Kosy_Tool\WObj:=Kosy_wobj;
    MoveJ Target_1090,v500,z100,Kosy_Tool\WObj:=Kosy_wobj;
    MoveJ Target_1100,v500,z100,Kosy_Tool\WObj:=Kosy_wobj;
    MoveJ Target_1110,v500,z100,Kosy_Tool\WObj:=Kosy_wobj;
    MoveJ Target_1120,v500,z100,Kosy_Tool\WObj:=Kosy_wobj;
    MoveL Target_1130,v600,z100,Kosy_Tool\WObj:=Kosy_wobj;
    MoveL Target_1140,v600,z100,Kosy_Tool\WObj:=Kosy_wobj;
    MoveJ Target_1150,v600,z100,Kosy_Tool\WObj:=Kosy_wobj;
    MoveJ Target_1160,v600,z100,Kosy_Tool\WObj:=Kosy_wobj;
    MoveL Target_1170,v1000,z100,Kosy_Tool\WObj:=Kosy_wobj;
  ENDPROC
  PROC Picktool()
    MoveJ Target_1290,v600,z100,Kosy_Tool\WObj:=Kosy_wobj;
    MoveL Target_1210,v600,z100,Kosy_Tool\WObj:=Kosy_wobj;
    MoveL Target_1200,v600,z100,Kosy_Tool\WObj:=Kosy_wobj;
    MoveL Target_1190,v600,z100,Kosy_Tool\WObj:=Kosy_wobj;
    MoveL Target_1180,v600,z100,Kosy_Tool\WObj:=Kosy_wobj;
  ENDPROC
  PROC Droptool()
    MoveJ Target_1220,v600,z100,Kosy_Tool\WObj:=Kosy_wobj;
    MoveL Target_1230,v600,z100,Kosy_Tool\WObj:=Kosy_wobj;
    MoveL Target_1240,v600,z100,Kosy_Tool\WObj:=Kosy_wobj;
    MoveL Target_1250,v600,z100,Kosy_Tool\WObj:=Kosy_wobj;
    MoveL Target_1260,v600,z100,Kosy_Tool\WObj:=Kosy_wobj;
    MoveL Target_1270,v1000,z100,Kosy_Tool\WObj:=Kosy_wobj;
    MoveL Target_1280,v1000,z100,Kosy_Tool\WObj:=Kosy_wobj;
  ENDPROC
ENDMODULE

